Omron CX-Programmer project NewProject (CX-Programmer 9.61)

# PLC NewPLC1: CP1E E20

## Global symbols (name address type ; comment)
0.00 BOOL  ; START
0.01 BOOL  ; E-STOP
0.02 BOOL  ; SENSOR 1
0.03 BOOL  ; SENSOR 2
0.04 BOOL  ; SENSOR 3
0.05 BOOL  ; SENSOR 4
0.06 BOOL  ; STOP
100.00 BOOL  ; SISTEM AKTIF
100.01 BOOL  ; CONVEYOR 1
100.02 BOOL  ; CONVEYOR 2
100.03 BOOL  ; MAGAZINE
100.04 BOOL  ; SILINDER 1
100.05 BOOL  ; SILINDER 2
100.06 BOOL  ; SILINDER 3

## Program NewProgram1 (cyclic task 0)

### Section Section1

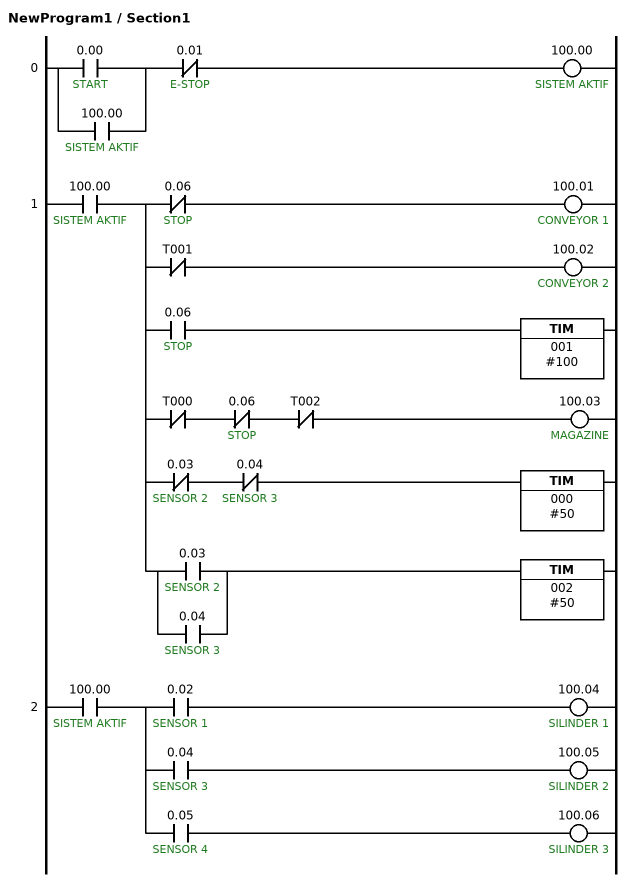
; rung 0
LD 0.00  ; START
OR 100.00  ; SISTEM AKTIF
ANDNOT 0.01  ; E-STOP
OUT 100.00  ; SISTEM AKTIF
; rung 1
LD 100.00  ; SISTEM AKTIF
OUT TR0
ANDNOT 0.06  ; STOP
OUT 100.01  ; CONVEYOR 1
LD TR0
ANDNOT T001
OUT 100.02  ; CONVEYOR 2
LD TR0
AND 0.06  ; STOP
TIM 001 #100
LD TR0
ANDNOT T000
ANDNOT 0.06  ; STOP
ANDNOT T002
OUT 100.03  ; MAGAZINE
LD TR0
ANDNOT 0.03  ; SENSOR 2
ANDNOT 0.04  ; SENSOR 3
TIM 000 #50
LD TR0
LD 0.03  ; SENSOR 2
OR 0.04  ; SENSOR 3
ANDLD
TIM 002 #50
; rung 2
LD 100.00  ; SISTEM AKTIF
OUT TR0
AND 0.02  ; SENSOR 1
OUT 100.04  ; SILINDER 1
LD TR0
AND 0.04  ; SENSOR 3
OUT 100.05  ; SILINDER 2
LD TR0
AND 0.05  ; SENSOR 4
OUT 100.06  ; SILINDER 3

### Section END
; rung 0
END(001)